DATA_BLOCK "FBD_Block_DB"
{ S7_Optimized_Access := 'TRUE' }
VERSION : 0.1
NON_RETAIN
"FBD_Block"

BEGIN

END_DATA_BLOCK

